TYPE ST_CommInfeedToLift :
STRUCT
	bReqExportProduct : BOOL; // Request lift to receive product from infeed.
	bBusyWithLift : BOOL; // Infeed busy with lift transfer (handshake/locking).
END_STRUCT
END_TYPE

(* stored: Version 1.1.0.1
   DUT ST_CommInfeedToLift: Id {1219a92a-d836-4077-8d49-bca1b0b8e0c8} *)
